(* IEC 61131-3 sources: cc_kush_rewrite/Functions, 19 files *)

(* ---- FC_Bunker_EmergencyStop.st ---- *)
FUNCTION FC_Bunker_EmergencyStop : BOOL
VAR_INPUT
	Bunker : ST_Bunker;
END_VAR
VAR
	j : INT;
END_VAR
// Остановка моторов вибраторов (4 шт на бункер)
FOR j := 1 TO 4 DO
	Bunker.MotorVibrator[j].qxKM_Power := FALSE;
	Bunker.MotorVibrator[j].VFD.qxStart := FALSE;
	Bunker.MotorVibrator[j].VFD.Frequency.rTargetFrequency := 0.0;
	Bunker.MotorVibrator[j].VFD.qrOutFrequency := 0.0;
END_FOR

// Остановка моторов вибропитателей (2 шт на бункер)
FOR j := 1 TO 2 DO
	Bunker.MotorVibFeeder[j].qxKM_Power := FALSE;
	Bunker.MotorVibFeeder[j].VFD.qxStart := FALSE;
	Bunker.MotorVibFeeder[j].VFD.Frequency.rTargetFrequency := 0.0;
	Bunker.MotorVibFeeder[j].VFD.qrOutFrequency := 0.0;
END_FOR

// Установка красного сигнала светофора
FC_Bunker_SetLightColor(Bunker := Bunker, eColor := E_LightColor.RED);

END_FUNCTION

(* ---- FC_Bunker_GetErrorBunker.st ---- *)
FUNCTION FC_Bunker_GetErrorBunker : BOOL
VAR_INPUT
	Bunker : REFERENCE TO ST_Bunker;
END_VAR
VAR
END_VAR
FC_Bunker_GetErrorBunker :=
	FC_Bunker_GetErrorMotorVibFeeder(Bunker := Bunker)
	OR FC_Bunker_GetErrorMotorVibrator(motor := Bunker.MotorVibrator[1])
	OR FC_Bunker_GetErrorMotorVibrator(motor := Bunker.MotorVibrator[2])
	OR FC_Bunker_GetErrorMotorVibrator(motor := Bunker.MotorVibrator[3])
	OR FC_Bunker_GetErrorMotorVibrator(motor := Bunker.MotorVibrator[4]);

END_FUNCTION

(* ---- FC_Bunker_GetErrorMotorVibFeeder.st ---- *)
FUNCTION FC_Bunker_GetErrorMotorVibFeeder : BOOL
VAR_INPUT
	Bunker : REFERENCE TO ST_Bunker;
END_VAR
VAR
END_VAR
FC_Bunker_GetErrorMotorVibFeeder :=
		Bunker.MotorVibFeeder[1].VFD.xStateFailure // Ошибка ЧРП, полученная по дискретному входу
		OR Bunker.MotorVibFeeder[1].VFD.xStateFailureLocal // Ошибка ЧРП, полученная программным путём
		OR Bunker.MotorVibFeeder[1].VFD.fbRangeDiagnostic.qxCriticalActive // Критическое значение тока эл. двигателя
		OR NOT Bunker.MotorVibFeeder[1].fbStatorOverheat.qxSignal // Перегрев статора (1 - норма, 0 - перегрев)
		OR Bunker.MotorVibFeeder[1].fbRangeDiagnostic[1].qxCriticalActive // Критический уровень нагрева подпишникового узла 1
		OR Bunker.MotorVibFeeder[1].fbRangeDiagnostic[2].qxCriticalActive // Критический уровень нагрева подпишникового узла 2

		OR Bunker.MotorVibFeeder[2].VFD.xStateFailure // Ошибка ЧРП, полученная по дискретному входу
		OR Bunker.MotorVibFeeder[2].VFD.xStateFailureLocal // Ошибка ЧРП, полученная программным путём
		OR Bunker.MotorVibFeeder[2].VFD.fbRangeDiagnostic.qxCriticalActive // Критическое значение тока эл. двигателя
		OR NOT Bunker.MotorVibFeeder[2].fbStatorOverheat.qxSignal // Перегрев статора (1 - норма, 0 - перегрев)
		OR Bunker.MotorVibFeeder[2].fbRangeDiagnostic[1].qxCriticalActive // Критический уровень нагрева подпишникового узла 1
		OR Bunker.MotorVibFeeder[2].fbRangeDiagnostic[2].qxCriticalActive; // Критический уровень нагрева подпишникового узла 2

END_FUNCTION

(* ---- FC_Bunker_GetErrorMotorVibrator.st ---- *)
FUNCTION FC_Bunker_GetErrorMotorVibrator : BOOL
VAR_INPUT
	motor : REFERENCE TO ST_Motor;
END_VAR
VAR
END_VAR
FC_Bunker_GetErrorMotorVibrator := (
	motor.VFD.xStateFailure // Ошибка ЧРП, полученная по дискретному входу
	OR motor.VFD.xStateFailureLocal // Ошибка ЧРП, полученная программным путём
	OR motor.VFD.fbRangeDiagnostic.qxCriticalActive // Критическое значение тока эл. двигателя
);

END_FUNCTION

(* ---- FC_Conveyor_GetErrorMotor.st ---- *)
FUNCTION FC_Conveyor_GetErrorMotor : BOOL
VAR_INPUT
	motor : REFERENCE TO ST_MotorWithFeedback;
END_VAR
VAR
END_VAR
FC_Conveyor_GetErrorMotor := (
	motor.VFD.xStateFailure // Ошибка ЧРП, полученная по дискретному входу
	OR motor.VFD.xStateFailureLocal // Ошибка ЧРП, полученная программным путём
	OR motor.VFD.fbRangeDiagnostic.qxCriticalActive // Критическое значение тока эл. двигателя
	OR NOT motor.fbStatorOverheat.qxSignal // Перегрев статора (1 - норма, 0 - перегрев)
);

END_FUNCTION

(* ---- FC_Conveyor_GetErrorSensors.st ---- *)
FUNCTION FC_Conveyor_GetErrorSensors : BOOL
VAR_INPUT
	Conveyor : REFERENCE TO ST_ConveyorPrefabricated;
END_VAR
VAR
END_VAR
FC_Conveyor_GetErrorSensors := (
	// == МОДУЛИ ДИСКРЕТНОГО ВХОДА ==
	// Контроль схода ленты (1 - норма, 0 - стоп)
	NOT Conveyor.fbZQAlarm[1].qxSignal
	OR NOT Conveyor.fbZQAlarm[2].qxSignal
	OR NOT Conveyor.fbZQAlarm[3].qxSignal
	OR NOT Conveyor.fbZQAlarm[4].qxSignal
	// Кабель-троссовый выключатель (1 - норма, 0 - стоп)
	OR NOT Conveyor.fbHQ_IsOk[1].qxSignal
	OR NOT Conveyor.fbHQ_IsOk[2].qxSignal
	OR NOT Conveyor.fbHQ_IsOk[3].qxSignal
	OR NOT Conveyor.fbHQ_IsOk[4].qxSignal
	// Контроль ограждения барабана (1 - норма, 0 - ограждения нет)
	OR NOT Conveyor.fbSQ_IsOk[1].qxSignal
	OR NOT Conveyor.fbSQ_IsOk[2].qxSignal
	// Контроль заштыбовки (1 - норма, 0 - ограждения нет)
	OR NOT Conveyor.fbGS1.qxSignal
	// Контроль продольного разрыва ленты (1 - норма, 0 - разрыв)
	OR NOT Conveyor.fbYS1.qxSignal
	// Обнаружение металла (1 - обнаружение, 0 - нет)
	OR Conveyor.fbYE1.qxSignal
);

END_FUNCTION

(* ---- FC_Dumper_GetErrorCommon.st ---- *)
FUNCTION FC_Dumper_GetErrorCommon : BOOL
VAR_INPUT
	Dumper : REFERENCE TO ST_Dumper;
END_VAR
VAR
END_VAR
FC_Dumper_GetErrorCommon :=
	FC_Dumper_GetErrorSensors(Dumper := Dumper)
	OR FC_Conveyor_GetErrorMotor(motor := Dumper.MotorConveyor[1])
	OR FC_Conveyor_GetErrorMotor(motor := Dumper.MotorConveyor[2])
	OR FC_Conveyor_GetErrorMotor(motor := Dumper.MotorRotation[1])
	OR FC_Conveyor_GetErrorMotor(motor := Dumper.MotorRotation[2]);

END_FUNCTION

(* ---- FC_Dumper_GetErrorSensors.st ---- *)
FUNCTION FC_Dumper_GetErrorSensors : BOOL
VAR_INPUT
	Dumper : REFERENCE TO ST_Dumper;
END_VAR
VAR
END_VAR
FC_Dumper_GetErrorSensors := (
	// == МОДУЛИ ДИСКРЕТНОГО ВХОДА ==
	// Контроль схода ленты (1 - норма, 0 - стоп)
	NOT Dumper.fbZQAlarm[1].qxSignal
	OR NOT Dumper.fbZQAlarm[2].qxSignal
	OR NOT Dumper.fbZQAlarm[3].qxSignal
	OR NOT Dumper.fbZQAlarm[4].qxSignal
	// Кабель-троссовый выключатель (1 - норма, 0 - стоп)
	OR NOT Dumper.fbHQ_IsOk[1].qxSignal
	OR NOT Dumper.fbHQ_IsOk[2].qxSignal
	OR NOT Dumper.fbHQ_IsOk[3].qxSignal
	OR NOT Dumper.fbHQ_IsOk[4].qxSignal
	// Контроль ограждения барабана (1 - норма, 0 - ограждения нет)
	OR NOT Dumper.fbSQ_IsOk[1].qxSignal
	OR NOT Dumper.fbSQ_IsOk[2].qxSignal
	// Контроль заштыбовки (1 - норма, 0 - ограждения нет)
	OR NOT Dumper.fbGS1.qxSignal
	// Контроль продольного разрыва ленты (1 - норма, 0 - разрыв)
	OR NOT Dumper.fbYS1.qxSignal
);

END_FUNCTION

(* ---- FC_Get_ErrorCommon.st ---- *)
FUNCTION FC_Get_ErrorCommon : BOOL
VAR_INPUT
	Bunker1 : REFERENCE TO ST_Bunker;
	Bunker2 : REFERENCE TO ST_Bunker;
	Bunker3 : REFERENCE TO ST_Bunker;
	Conveyor : REFERENCE TO ST_ConveyorPrefabricated;
	Dumper : REFERENCE TO ST_Dumper;
END_VAR
VAR
END_VAR
FC_Get_ErrorCommon :=
	FC_Bunker_GetErrorBunker(Bunker := Bunker1) // Получение ошибки бункера 1
	OR FC_Bunker_GetErrorBunker(Bunker := Bunker2) // Получение ошибки бункера 2
	OR FC_Bunker_GetErrorBunker(Bunker := Bunker3) // Получение ошибки бункера 3
	OR FC_Conveyor_GetErrorCommon(Conveyor := Conveyor) // Получение ошибки сборного конвейера
	OR FC_Dumper_GetErrorCommon(Dumper := Dumper) // Получение ошибки отвалообразователя
	OR FC_Bunker_GetErrorWeight(Bunker1 := Bunker1, Bunker2 := Bunker2, Bunker3 := Bunker3); // Проверка заполненности бункеров

END_FUNCTION

(* ---- FC_ModbusReadBool.st ---- *)
// Чтение BOOL из бита Modbus регистра
// Возвращает TRUE при успешном чтении, FALSE при ошибке (неверный индекс бита)
FUNCTION FC_ModbusReadBool : BOOL
VAR_INPUT
    pRegisters : POINTER TO WORD;  // Указатель на массив Modbus регистров
    iRegisterIndex : INT;           // Индекс регистра
    iBitIndex : INT;                // Номер бита в регистре (0..15)
END_VAR
VAR_OUTPUT
    xValue : BOOL;                  // Прочитанное значение
END_VAR
VAR
    wMask : WORD;
    pTargetRegister : POINTER TO WORD;
END_VAR
    // Проверка диапазона индекса бита
    IF iBitIndex >= 0 AND iBitIndex <= 15 THEN
        // Вычислить адрес целевого регистра
        pTargetRegister := pRegisters + iRegisterIndex;

        // Создать маску для бита
        wMask := SHL(1, iBitIndex);

        // Прочитать бит
        xValue := (pTargetRegister^ AND wMask) <> 0;

        FC_ModbusReadBool := TRUE;  // Успех
    ELSE
        xValue := FALSE;
        FC_ModbusReadBool := FALSE;  // Ошибка: неверный индекс бита
    END_IF
END_FUNCTION

(* ---- FC_ModbusReadInt.st ---- *)
// Чтение INT из Modbus регистра
// Возвращает TRUE при успешном чтении
FUNCTION FC_ModbusReadInt : BOOL
VAR_INPUT
    pRegisters : POINTER TO WORD;  // Указатель на массив Modbus регистров
    iRegisterIndex : INT;           // Индекс регистра
END_VAR
VAR_OUTPUT
    iValue : INT;                   // Прочитанное значение
END_VAR
VAR
    pTargetRegister : POINTER TO WORD;
END_VAR
    // Вычислить адрес целевого регистра и прочитать значение
    pTargetRegister := pRegisters + iRegisterIndex*2;
    iValue := WORD_TO_INT(pTargetRegister^);
    FC_ModbusReadInt := TRUE;

END_FUNCTION

(* ---- FC_ModbusReadReal.st ---- *)
// Чтение REAL из 2 последовательных Modbus регистров через UNION
// Возвращает TRUE при успешном чтении
// REAL (32 бита) читается из 2 регистров (по 16 бит каждый)
FUNCTION FC_ModbusReadReal : BOOL
VAR_INPUT
    pRegisters : POINTER TO WORD;  // Указатель на массив Modbus регистров
    iRegisterIndex : INT;           // Начальный индекс (читает 2 регистра: N и N+1)
END_VAR
VAR_OUTPUT
    rValue : REAL;                  // Прочитанное значение
END_VAR
VAR
    uConverter : U_RealToWord;
    pTargetRegister : POINTER TO WORD;
END_VAR
    // Чтение первого регистра (младшее слово)
    pTargetRegister := pRegisters + iRegisterIndex;
    uConverter.wTag[0] := pTargetRegister^;

    // Чтение второго регистра (старшее слово)
    pTargetRegister := pTargetRegister + 1;
    uConverter.wTag[1] := pTargetRegister^;

    // Преобразовать в REAL
    rValue := uConverter.rTag;

    FC_ModbusReadReal := TRUE;
END_FUNCTION

(* ---- FC_ModbusReadTime.st ---- *)
// Чтение TIME из 2 последовательных Modbus регистров через UNION
// Возвращает TRUE при успешном чтении
// TIME (32 бита) читается из 2 регистров (по 16 бит каждый)
FUNCTION FC_ModbusReadTime : BOOL
VAR_INPUT
    pRegisters : POINTER TO WORD;  // Указатель на массив Modbus регистров
    iRegisterIndex : INT;           // Начальный индекс (читает 2 регистра: N и N+1)
END_VAR
VAR_OUTPUT
    tValue : TIME;                  // Прочитанное значение
END_VAR
VAR
    uConverter : U_TimeToWord;
    pTargetRegister : POINTER TO WORD;
END_VAR
    // Чтение первого регистра (младшее слово)
    pTargetRegister := pRegisters + iRegisterIndex*2;
    uConverter.wTag[1] := pTargetRegister^;

    // Чтение второго регистра (старшее слово)
    pTargetRegister := pTargetRegister + 2;
    uConverter.wTag[0] := pTargetRegister^;

    // Преобразовать в TIME
    tValue := uConverter.tTag;

    FC_ModbusReadTime := TRUE;

END_FUNCTION

(* ---- FC_ModbusWriteBool.st ---- *)
// Запись BOOL в бит Modbus регистра
// Возвращает TRUE при успешной записи, FALSE при ошибке (неверный индекс бита)
FUNCTION FC_ModbusWriteBool : BOOL
VAR_INPUT
    pRegisters : POINTER TO WORD;  // Указатель на массив Modbus регистров
    iRegisterIndex : INT;           // Индекс регистра
    iBitIndex : INT;                // Номер бита в регистре (0..15)
    xValue : BOOL;                  // Значение для записи
END_VAR
VAR
    wMask : WORD;
    pTargetRegister : POINTER TO WORD;
END_VAR
    // Проверка диапазона индекса бита
    IF iBitIndex >= 0 AND iBitIndex <= 15 THEN
        // Вычислить адрес целевого регистра
        pTargetRegister := pRegisters + iRegisterIndex*2;

        wMask := SHL(1, iBitIndex);  // Создать маску для бита

        IF xValue THEN
            // Установить бит (OR)
            pTargetRegister^ := pTargetRegister^ OR wMask;
        ELSE
            // Сбросить бит (AND NOT)
            pTargetRegister^ := pTargetRegister^ AND NOT wMask;
        END_IF

        FC_ModbusWriteBool := TRUE;  // Успех
    ELSE
        FC_ModbusWriteBool := FALSE;  // Ошибка: неверный индекс бита
    END_IF

END_FUNCTION

(* ---- FC_ModbusWriteInt.st ---- *)
// Запись INT в Modbus регистр
// Возвращает TRUE при успешной записи
FUNCTION FC_ModbusWriteInt : BOOL
VAR_INPUT
    pRegisters : POINTER TO WORD;  // Указатель на массив Modbus регистров
    iRegisterIndex : INT;           // Индекс регистра
    iValue : INT;                   // Значение для записи
END_VAR
VAR
    pTargetRegister : POINTER TO WORD;
END_VAR
    // Вычислить адрес целевого регистра и записать значение
    pTargetRegister := pRegisters + iRegisterIndex*2;
    pTargetRegister^ := INT_TO_WORD(iValue);
    FC_ModbusWriteInt := TRUE;

END_FUNCTION

(* ---- FC_ModbusWriteReal.st ---- *)
// Запись REAL в 2 последовательных Modbus регистра через UNION
// Возвращает TRUE при успешной записи
// REAL (32 бита) упаковывается в 2 регистра (по 16 бит каждый)
FUNCTION FC_ModbusWriteReal : BOOL
VAR_INPUT
    pRegisters : POINTER TO WORD;  // Указатель на массив Modbus регистров
    iRegisterIndex : INT;           // Начальный индекс (занимает 2 регистра: N и N+1)
    rValue : REAL;                  // Значение для записи
END_VAR
VAR
    uConverter : U_RealToWord;
    pTargetRegister : POINTER TO WORD;
END_VAR
    uConverter.rTag := rValue;

    // Запись первого регистра (младшее слово)
    pTargetRegister := pRegisters + iRegisterIndex;
    pTargetRegister^ := uConverter.wTag[0];

    // Запись второго регистра (старшее слово)
    pTargetRegister := pTargetRegister + 1;
    pTargetRegister^ := uConverter.wTag[1];

    FC_ModbusWriteReal := TRUE;
END_FUNCTION

(* ---- FC_ModbusWriteTime.st ---- *)
// Запись TIME в 2 последовательных Modbus регистра через UNION
// Возвращает TRUE при успешной записи
// TIME (32 бита) упаковывается в 2 регистра (по 16 бит каждый)
FUNCTION FC_ModbusWriteTime : BOOL
VAR_INPUT
    pRegisters : POINTER TO WORD;  // Указатель на массив Modbus регистров
    iRegisterIndex : INT;           // Начальный индекс (занимает 2 регистра: N и N+1)
    tValue : TIME;                  // Значение для записи
END_VAR
VAR
    uConverter : U_TimeToWord;
    pTargetRegister : POINTER TO WORD;
END_VAR
    uConverter.tTag := tValue;

    // Запись первого регистра (младшее слово)
    pTargetRegister := pRegisters + iRegisterIndex*2;
    pTargetRegister^ := uConverter.wTag[1];

    // Запись второго регистра (старшее слово)
    pTargetRegister := pTargetRegister + 2;
    pTargetRegister^ := uConverter.wTag[0];

    FC_ModbusWriteTime := TRUE;

END_FUNCTION

(* ---- FC_SwapBytesInWordArray.st ---- *)
FUNCTION FC_SwapBytesInWordArray : ARRAY [0..1] OF WORD
VAR_INPUT
    awInputArray : ARRAY [0..1] OF WORD;        // Входной массив из двух WORD
END_VAR
VAR
    uByteConverter : U_ByteToWord;              // Конвертер для работы с байтами
    awOutputArray : ARRAY [0..1] OF WORD;       // Выходной массив
END_VAR

// Обработка первого WORD (индекс 0)
uByteConverter.wTag := awInputArray[0];
// Меняем местами байты и записываем в выходной массив
awOutputArray[0] := SHL(TO_WORD(uByteConverter.bTag[0]), 8) OR TO_WORD(uByteConverter.bTag[1]);

// Обработка второго WORD (индекс 1)
uByteConverter.wTag := awInputArray[1];
// Меняем местами байты и записываем в выходной массив
awOutputArray[1] := SHL(TO_WORD(uByteConverter.bTag[0]), 8) OR TO_WORD(uByteConverter.bTag[1]);

// Возвращаем преобразованный массив
FC_SwapBytesInWordArray := awOutputArray;

END_FUNCTION

(* ---- FC_VFD_ChangeReadMode.st ---- *)
FUNCTION FC_VFD_ChangeReadMode : BOOL
VAR_INPUT
	vfd : REFERENCE TO ST_VFD;
	mode : BOOL; // 0 - физический вход, 1 - Modbus
END_VAR
VAR
END_VAR
IF mode THEN
	vfd.rActualFrequency := vfd.uActualFrequency.rTag; // Чтение регистров ModbusRTU
ELSE
	vfd.rActualFrequency := vfd.fbActualFrequency.qrProcessedValue; // Чтение обработанного (масштабированного) аналогового сигнала с модуля
END_IF;

END_FUNCTION
